TYPE ST_KVM_App :
STRUCT
	wSID	: WORD:=1;	
	wAID	: WORD:=1;	
	sCID	: STRING(8):='12345678';
	sName	: STRING(63);	
	sInfo	: STRING(255);
END_STRUCT
END_TYPE

(* stored: Version 1.1.0.1, ProductVersion 3.1.4024.12
   DUT ST_KVM_App: Id {f25fadf0-4c2b-4c46-9b14-13c48085c92d} *)
